// Mitsubishi GX Works2 project: Project - Done   PLC: FX3G

// global labels: Global1
VAR_GLOBAL
  startDay AT X007 : BOOL;
  startDayLamp AT Y007 : BOOL;
  amounts AT M0 : BOOL;
END_VAR
VAR_GLOBAL CONSTANT
  whippedCream : REAL := 300.0;
END_VAR
VAR_GLOBAL
  CreamTank AT D1105 : REAL;
END_VAR
VAR_GLOBAL CONSTANT
  Chocolate : REAL := 240;
  Chocolate_input : REAL := 240;
  whippedCream_input : REAL := 300;
END_VAR
VAR_GLOBAL
  ChocolateTank AT D1101 : REAL;
END_VAR
VAR_GLOBAL CONSTANT
  Biscuit_input : REAL := 6;
END_VAR
VAR_GLOBAL
  BiscuitTank AT D1103 : REAL;
  start_Proccessing AT X011 : BOOL;
END_VAR
VAR_GLOBAL CONSTANT
  Const_6 : REAL := 6;
END_VAR
VAR_GLOBAL
  binary_Less_than_6 AT M1 : BOOL;
END_VAR
VAR_GLOBAL CONSTANT
  Const_300 : REAL := 300;
END_VAR
VAR_GLOBAL
  binary_Less_than_300 AT M2 : BOOL;
END_VAR
VAR_GLOBAL CONSTANT
  Const_0 : REAL;
END_VAR
VAR_GLOBAL
  No_More_Raw AT M3 : BOOL;
  No_More_Raw_B AT M3 : BOOL;
  No_More_Raw_C AT M4 : BOOL;
  Proccess_B_Tank AT D1103 : REAL;
  Proccess_C_Tank AT D1104 : REAL;
  machine_A_On AT X010 : BOOL;
  machine_A_still_On AT M0 : BOOL;
  turn_machine_A_off AT X005 : BOOL;
  sen_Surface AT X001 : BOOL;
  sen_30 AT X002 : BOOL;
  sen_15 AT X003 : BOOL;
  currrently_sprinkling AT Y004 : BOOL;
  sen_camera AT X004 : BOOL;
END_VAR
VAR_GLOBAL CONSTANT
  TC0 : INT := 40;
  TC1 : INT := 40;
  constant_sec_4 : INT := 5;
END_VAR
VAR_GLOBAL
  time_total_4_sec_end_movement AT TC0 : BOOL;
  timer_ts0 AT TS0 : BOOL;
  lamp0 AT Y000 : BOOL;
  input_for_blinking AT M4 : BOOL;
  time_total_4_sec_end_movement2 AT TC1 : BOOL;
  timer_ts1 AT TS1 : BOOL;
  lamp1 AT Y001 : BOOL;
END_VAR
VAR_GLOBAL CONSTANT
  const_zero_val_word : INT;
END_VAR
VAR_GLOBAL
  analog_output AT D8282 : INT;
END_VAR
VAR_GLOBAL CONSTANT
  Const_240 : REAL := 240;
END_VAR
VAR_GLOBAL
  binary_Less_than_240 AT M3 : BOOL;
END_VAR
VAR_GLOBAL CONSTANT
  constant_4_sec : INT := 40;
END_VAR
VAR_GLOBAL
  time_total_4_sec_end_movement3 AT TC3 : BOOL;
END_VAR
VAR_GLOBAL CONSTANT
  constant_half_sec : INT := 5;
END_VAR
VAR_GLOBAL
  timer_ts3 AT TS3 : BOOL;
  start_Frosting AT X006 : BOOL;
  analog_Input_1 AT D8280 : INT;
  save_Analog_Value AT D1134 : INT;
  value_Sampled AT M10 : BOOL;
END_VAR
VAR_GLOBAL CONSTANT
  analog_upper_bound : INT := 3900;
  upper_bound_analog_value : INT := 3510;
  analog_lower_value : INT := 390;
END_VAR
VAR_GLOBAL
  input_is_invalid AT M11 : BOOL;
  currently_frosting AT Y003 : BOOL;
END_VAR
VAR_GLOBAL CONSTANT
  single_frosting_check : INT := 1950;
END_VAR
VAR_GLOBAL
  single_frosting AT M12 : BOOL;
  double_frosting AT M13 : BOOL;
END_VAR
VAR_GLOBAL CONSTANT
  chocalate_single_amount : INT := 120;
END_VAR
VAR_GLOBAL
  dipping_tank AT D1107 : REAL;
END_VAR
VAR_GLOBAL CONSTANT
  chocalate_double_amount : INT := 240;
END_VAR
VAR_GLOBAL
  frostimg_time AT TC5 : BOOL;
END_VAR
VAR_GLOBAL CONSTANT
  const_5_sec : INT := 50;
END_VAR
VAR_GLOBAL
  frosting_time_over AT TS5 : BOOL;
END_VAR
VAR_GLOBAL CONSTANT
  const_chocalate_single_amount : REAL := 120;
  const_chocalate_double_amount : REAL := 240;
END_VAR
VAR_GLOBAL
  analog_Input_2 AT D8281 : INT;
  start_Packing AT X011 : BOOL;
END_VAR
VAR_GLOBAL CONSTANT
  const_count_5 : INT := 5;
END_VAR
VAR_GLOBAL
  start_packing_counter AT CC1 : BOOL;
  finish_packing_5_counter AT CS1 : BOOL;
  packing_5_lamp AT Y002 : BOOL;
  end_of_movment AT M20 : BOOL;
  pack_one_krembo AT X000 : BOOL;
  finish_packing_counter AT CC2 : BOOL;
END_VAR
VAR_GLOBAL CONSTANT
  const_count_1 : INT := 1;
END_VAR
VAR_GLOBAL
  finish_packing_6_counter AT CS3 : BOOL;
  finish_packing_1_counter AT CS2 : BOOL;
  finish_total_packing_counter AT CC3 : BOOL;
END_VAR
VAR_GLOBAL CONSTANT
  const_count_6 : INT := 6;
END_VAR
VAR_GLOBAL
  finish_packing_all_counter AT CS3 : BOOL;
  Proccess_Cream_Tank AT D1109 : REAL;
  Proccess_chocolate_tank AT D1107 : REAL;
  end_of_packing AT M22 : BOOL;
END_VAR
VAR_GLOBAL CONSTANT
  Const_6_krembos : REAL := 240;
END_VAR
VAR_GLOBAL
  krembo_total_count AT D10 : REAL;
  word_krembo_total AT D1150 : INT;
END_VAR
VAR_GLOBAL CONSTANT
  Const_6_x : REAL := 2340;
END_VAR
VAR_GLOBAL
  double_frosting_lamp AT M100 : BOOL;
  stsrt_frosting_lamp AT M21 : BOOL;
  start_frosting_lamp AT M21 : BOOL;
  frosting AT M34 : BOOL;
  krembo_added AT M40 : BOOL;
  less_Than_6 AT M41 : BOOL;
  cream_less_than_300 AT M42 : BOOL;
  chocolate_less_than_240 AT M43 : BOOL;
  biscuit_less_Than_6 AT M41 : BOOL;
END_VAR
VAR_GLOBAL CONSTANT
  double_frosting_check : INT := 2340;
END_VAR
VAR_GLOBAL
  converted AT M45 : BOOL;
  time_total_3_sec_end_day : BOOL;
  time_total_3_sec_end_day2 : BOOL;
  timer_ts100 : BOOL;
  timer_ts101 : BOOL;
  const_3_sec_timer AT TC6 : BOOL;
END_VAR
VAR_GLOBAL CONSTANT
  const_3_sec : INT := 30;
END_VAR
VAR_GLOBAL
  time_3_sec AT TC6 : BOOL;
  timer_ts_6 AT TS6 : BOOL;
  time_3_sec_end_day AT TC7 : BOOL;
  day_over_lamp AT M46 : BOOL;
  day_over AT M46 : BOOL;
  timer_ts_7 AT TS7 : BOOL;
  time_3_sec_end_day2 AT TC8 : BOOL;
  end_Day_Blink AT M50 : BOOL;
  timer_ts_8 AT TS8 : BOOL;
  fake_light AT M51 : BOOL;
  input_for_end_day_blink AT M60 : BOOL;
  flick_time_still AT M70 : BOOL;
  flicker_end_day AT M71 : BOOL;
  blink_1 AT M72 : BOOL;
  tc_blink1 AT TC9 : BOOL;
END_VAR
VAR_GLOBAL CONSTANT
  const_quick_3 : INT := 5;
END_VAR
VAR_GLOBAL
  ts_blink1 AT TS9 : BOOL;
  za_blink1 AT M73 : BOOL;
  tc_blink2 AT TC10 : BOOL;
  ts_blink10 AT TS10 : BOOL;
  za_blink2 AT M74 : BOOL;
  ts_blink2 AT TS10 : BOOL;
END_VAR

// task Task_01 (event TRUE, interval 0, priority 31): POU_01

PROGRAM POU_01
VAR
  timer_ts6 : BOOL;
END_VAR
(* structured ladder/FBD written out as ST: instructions are called as NAME(EN, inputs, outputs); _pN, _eN, _tN stand for wires *)
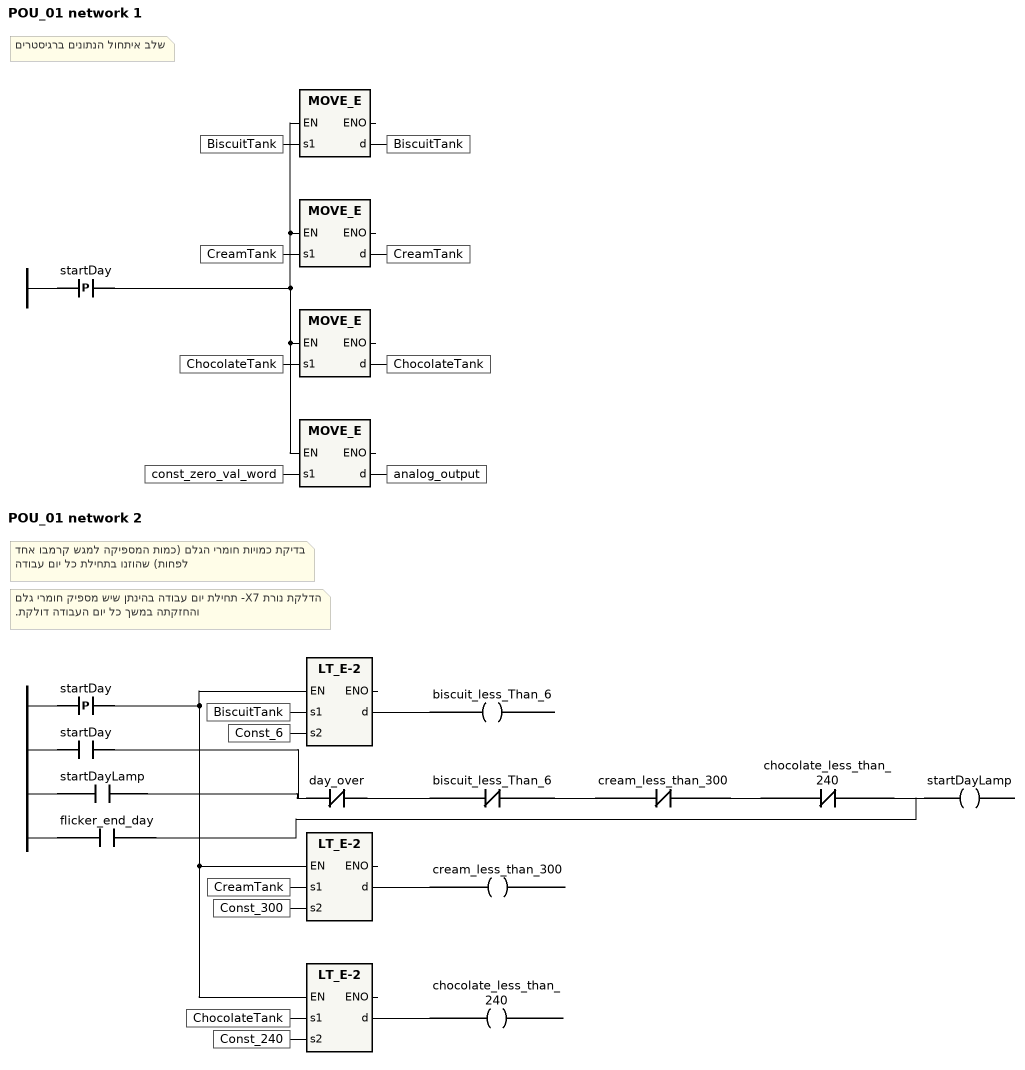
(* network 1 User input *)
(* שלב איתחול הנתונים ברגיסטרים *)
_p1 := LDP(TRUE, startDay);
MOVE_E(_p1, BiscuitTank, BiscuitTank);
MOVE_E(_p1, CreamTank, CreamTank);
MOVE_E(_p1, ChocolateTank, ChocolateTank);
MOVE_E(_p1, const_zero_val_word, analog_output);
(* network 2 Day initialize *)
(* בדיקת כמויות חומרי הגלם (כמות המספיקה למגש קרמבו אחד לפחות) שהוזנו בתחילת כל יום עבודה *)
(* הדלקת נורת X7- תחילת יום עבודה בהינתן שיש מספיק חומרי גלם והחזקתה במשך כל יום העבודה דולקת. *)
_p1 := LDP(TRUE, startDay);
LT_E(_p1, BiscuitTank, Const_6, _t2);
biscuit_less_Than_6 := _t2;
LT_E(_p1, CreamTank, Const_300, _t3);
cream_less_than_300 := _t3;
LT_E(_p1, ChocolateTank, Const_240, _t4);
chocolate_less_than_240 := _t4;
startDayLamp := (((((startDay OR startDayLamp) AND NOT day_over) AND NOT biscuit_less_Than_6) AND NOT cream_less_than_300) AND NOT chocolate_less_than_240) OR flicker_end_day;
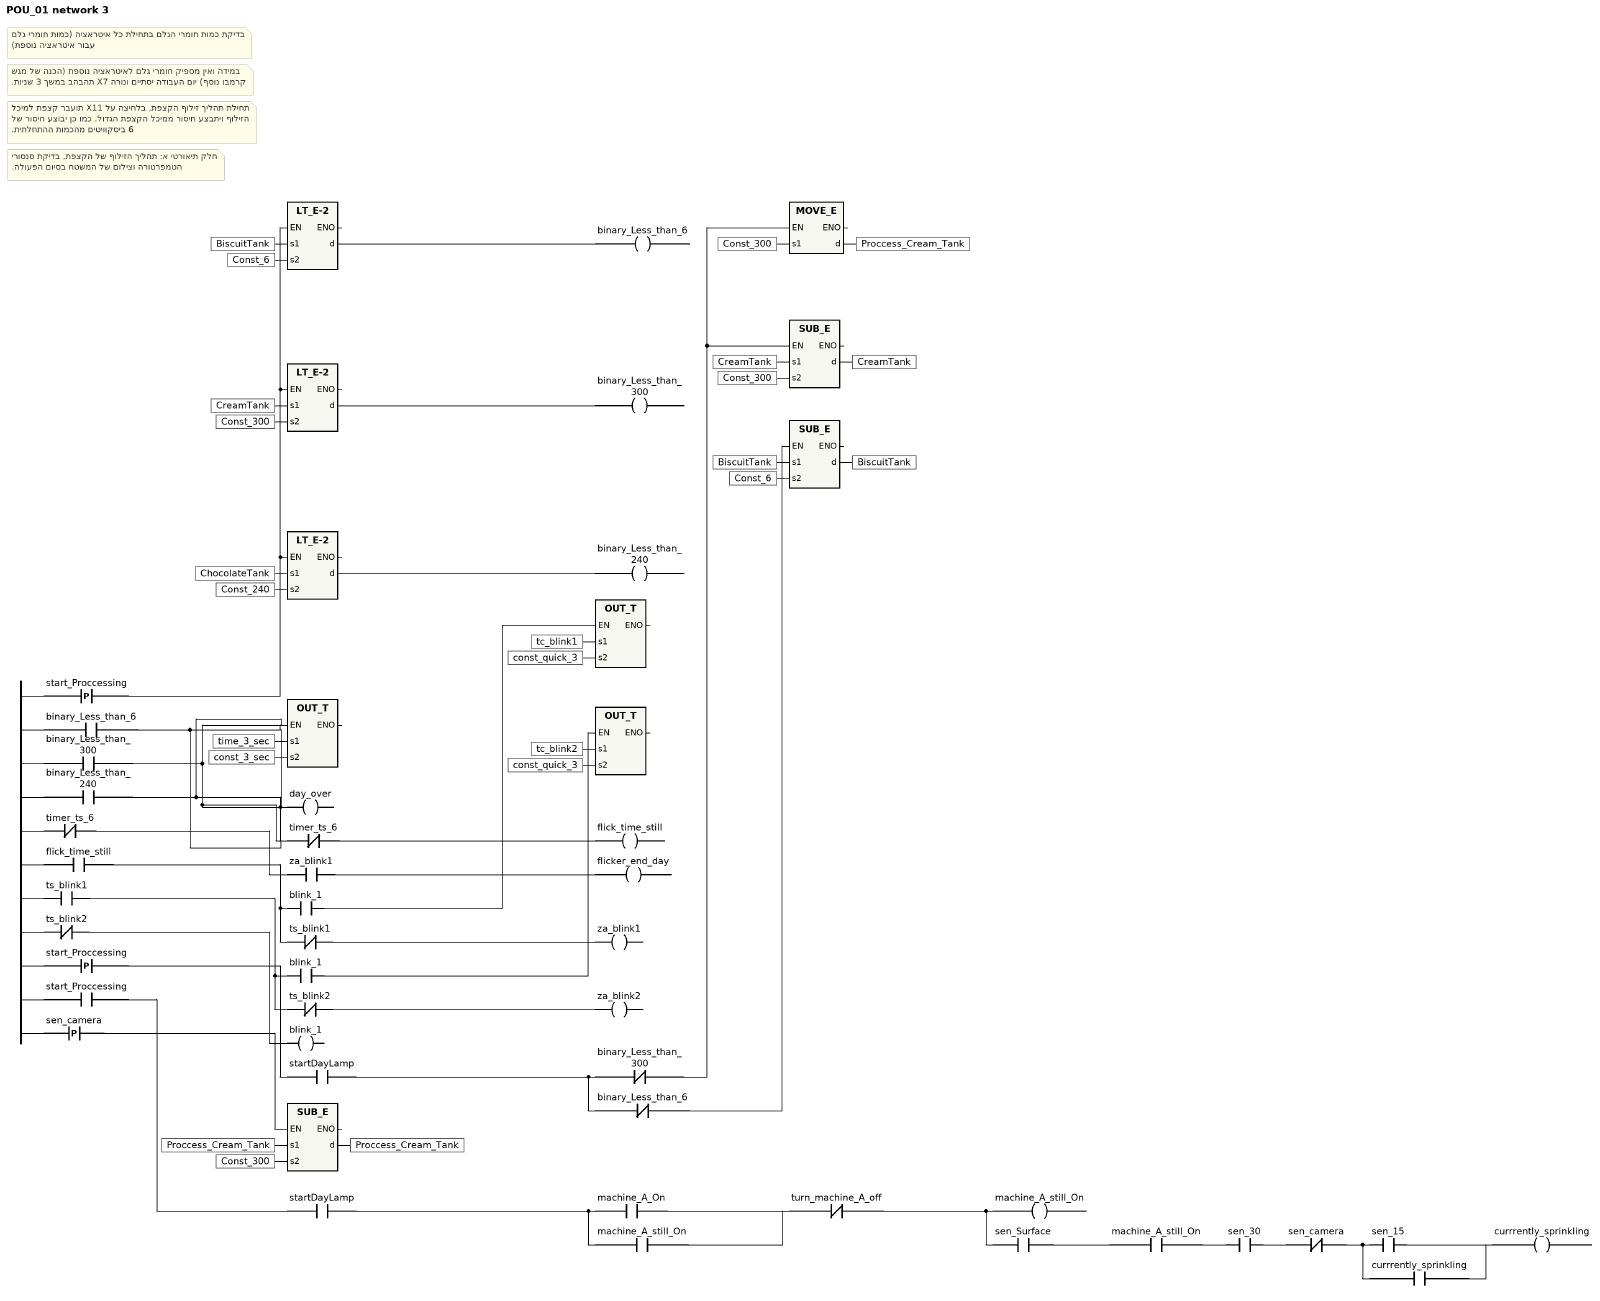
(* network 3 Whipping Cream Proc *)
(* בדיקת כמות חומרי הגלם בתחילת כל איטראציה (כמות חומרי גלם עבור איטראציה נוספת) *)
(* במידה ואין מספיק חומרי גלם לאיטראציה נוספת (הכנה של מגש קרמבו נוסף) יום העבודה יסתיים ונורה X7 תהבהב במשך 3 שניות. *)
(* תחילת תהליך זילוף הקצפת, בלחיצה על X11 תועבר קצפת למיכל הזילוף ויתבצע חיסור ממיכל הקצפת הגדול. כמו כן יבוצע חיסור של 6 ביסקוויטים מהכמות ההתחלתית. *)
(* חלק תיאורטי א: תהליך הזילוף של הקצפת, בדיקת סנסורי הטמפרטורה וצילום של המשטח בסיום הפעולה. *)
_p1 := LDP(TRUE, start_Proccessing);
LT_E(_p1, BiscuitTank, Const_6, _t2);
binary_Less_than_6 := _t2;
LT_E(_p1, CreamTank, Const_300, _t3);
binary_Less_than_300 := _t3;
LT_E(_p1, ChocolateTank, Const_240, _t4);
binary_Less_than_240 := _t4;
_p5 := binary_Less_than_6 OR binary_Less_than_300 OR binary_Less_than_240;
OUT_T(_p5, time_3_sec, const_3_sec);
day_over := _p5;
flick_time_still := _p5 AND NOT timer_ts_6;
flicker_end_day := NOT timer_ts_6 AND za_blink1;
OUT_T(flick_time_still AND blink_1, tc_blink1, const_quick_3);
za_blink1 := flick_time_still AND NOT ts_blink1;
OUT_T(ts_blink1 AND blink_1, tc_blink2, const_quick_3);
za_blink2 := ts_blink1 AND NOT ts_blink2;
blink_1 := NOT ts_blink2;
_p6 := LDP(TRUE, start_Proccessing) AND startDayLamp;
_p7 := _p6 AND NOT binary_Less_than_300;
MOVE_E(_p7, Const_300, Proccess_Cream_Tank);
SUB_E(_p7, CreamTank, Const_300, CreamTank);
SUB_E(_p6 AND NOT binary_Less_than_6, BiscuitTank, Const_6, BiscuitTank);
_p8 := start_Proccessing AND startDayLamp;
_p9 := ((_p8 AND machine_A_On) OR (_p8 AND machine_A_still_On)) AND NOT turn_machine_A_off;
machine_A_still_On := _p9;
_p10 := _p9 AND sen_Surface AND machine_A_still_On AND sen_30 AND NOT sen_camera;
currrently_sprinkling := (_p10 AND sen_15) OR (_p10 AND currrently_sprinkling);
SUB_E(LDP(TRUE, sen_camera), Proccess_Cream_Tank, Const_300, Proccess_Cream_Tank);
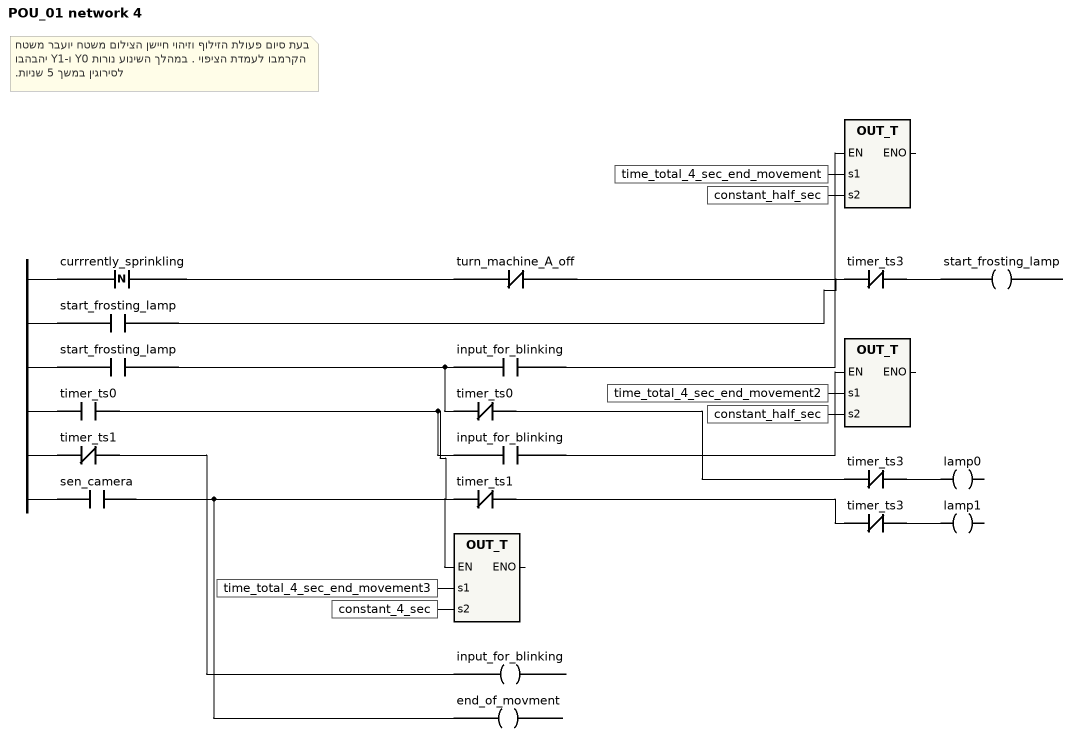
(* network 4 Move the krembo to B *)
(* בעת סיום פעולת הזילוף וזיהוי חיישן הצילום משטח יועבר משטח הקרמבו לעמדת הציפוי . במהלך השינוע נורות Y0 ו-Y1 יהבהבו לסירוגין במשך 5 שניות. *)
start_frosting_lamp := ((LDF(TRUE, currrently_sprinkling) AND NOT turn_machine_A_off) OR start_frosting_lamp) AND NOT timer_ts3;
OUT_T(start_frosting_lamp AND input_for_blinking, time_total_4_sec_end_movement, constant_half_sec);
lamp0 := start_frosting_lamp AND NOT timer_ts0 AND NOT timer_ts3;
OUT_T(timer_ts0 AND input_for_blinking, time_total_4_sec_end_movement2, constant_half_sec);
lamp1 := timer_ts0 AND NOT timer_ts1 AND NOT timer_ts3;
input_for_blinking := NOT timer_ts1;
OUT_T(sen_camera, time_total_4_sec_end_movement3, constant_4_sec);
end_of_movment := sen_camera;
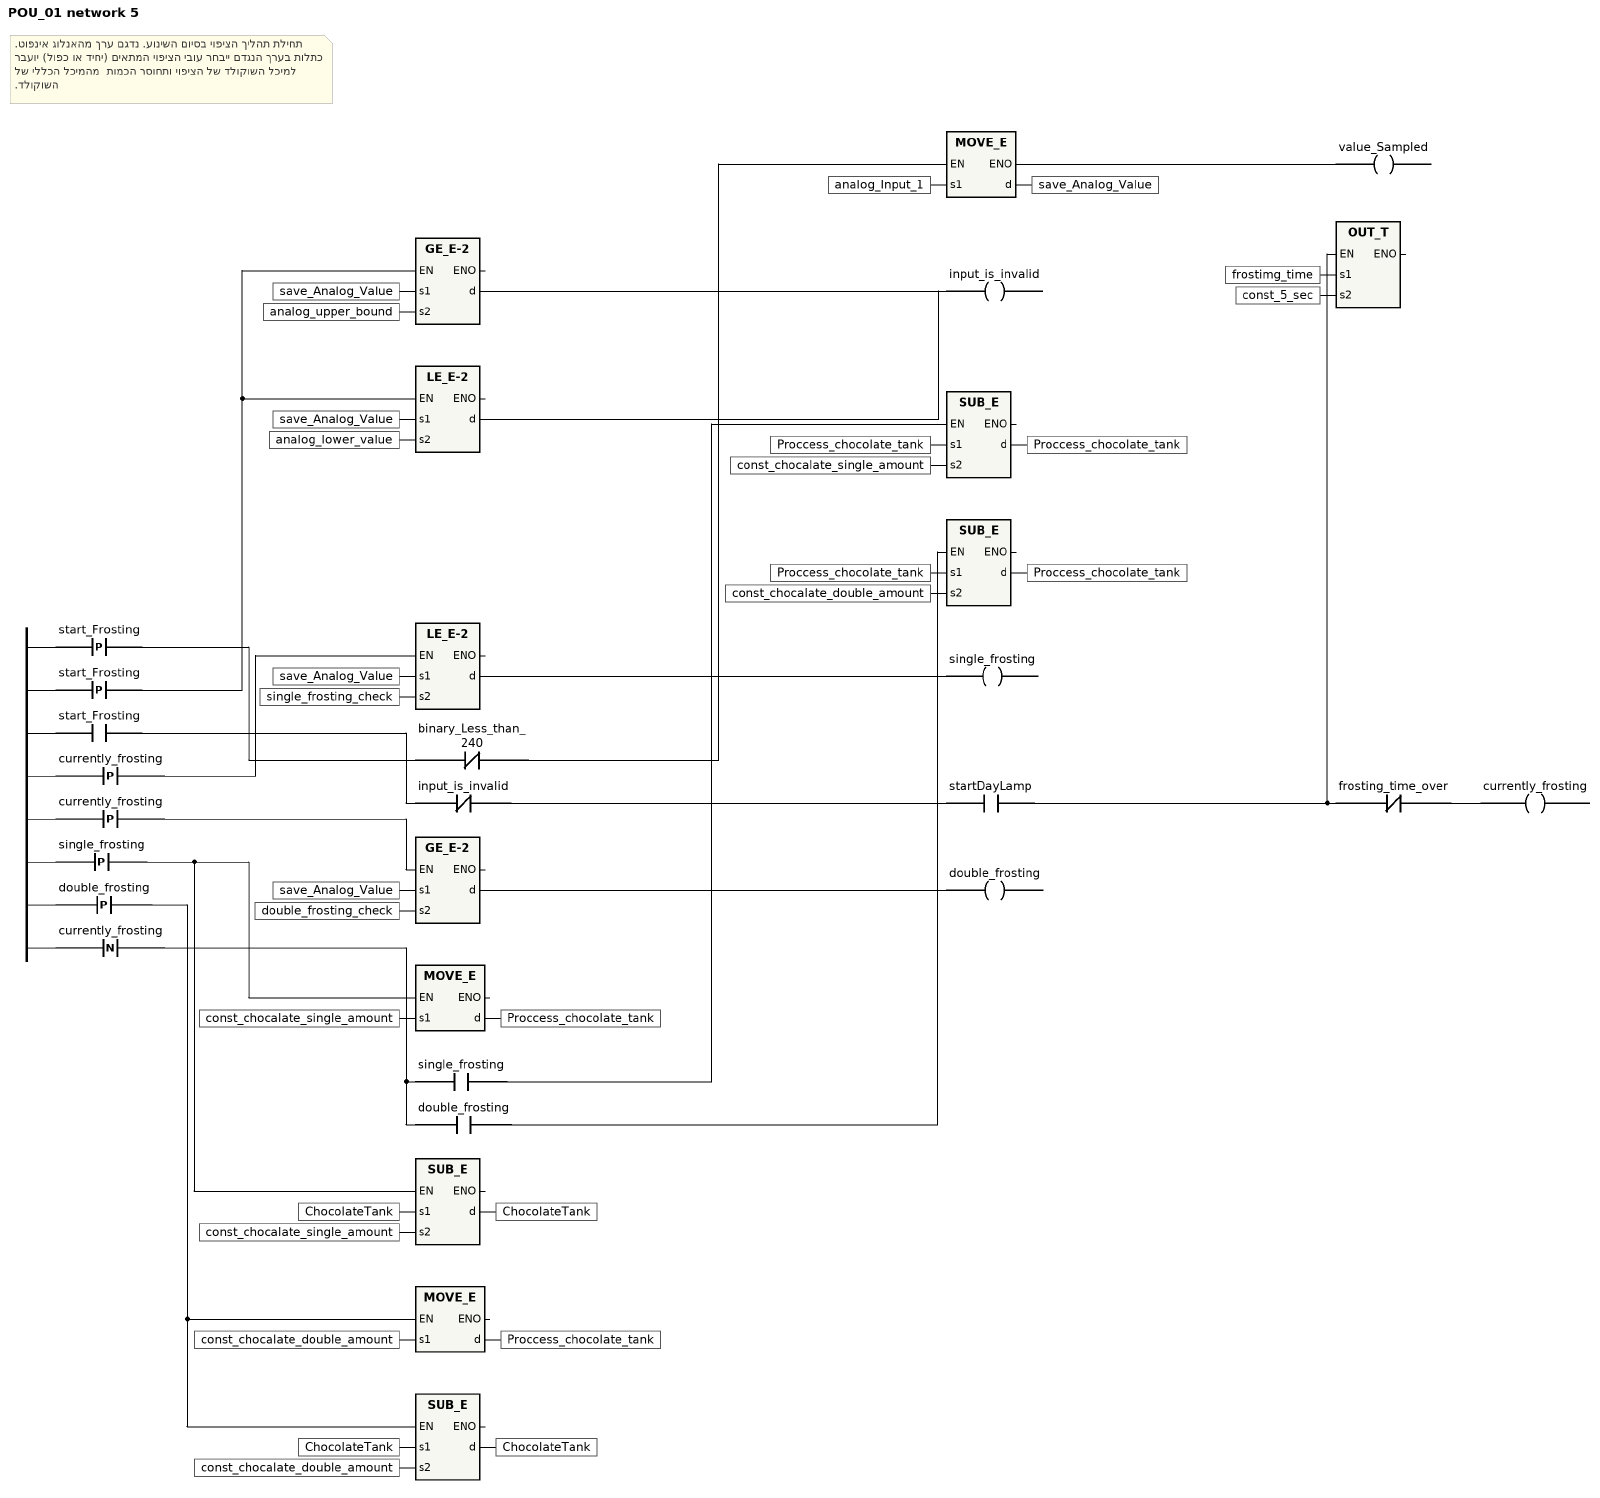
(* network 5 Frosting *)
(* תחילת תהליך הציפוי בסיום השינוע. נדגם ערך מהאנלוג אינפוט. כתלות בערך הנגדם ייבחר עובי הציפוי המתאים (יחיד או כפול) יועבר למיכל השוקולד של הציפוי ותחוסר הכמות  מהמיכל הכללי של השוקולד. *)
_e1 := MOVE_E(LDP(TRUE, start_Frosting) AND NOT binary_Less_than_240, analog_Input_1, save_Analog_Value);
value_Sampled := _e1;
_p2 := LDP(TRUE, start_Frosting);
GE_E(_p2, save_Analog_Value, analog_upper_bound, _t3);
LE_E(_p2, save_Analog_Value, analog_lower_value, _t4);
input_is_invalid := _t3 OR _t4;
_p5 := start_Frosting AND NOT input_is_invalid AND startDayLamp;
OUT_T(_p5, frostimg_time, const_5_sec);
currently_frosting := _p5 AND NOT frosting_time_over;
LE_E(LDP(TRUE, currently_frosting), save_Analog_Value, single_frosting_check, _t6);
single_frosting := _t6;
GE_E(LDP(TRUE, currently_frosting), save_Analog_Value, double_frosting_check, _t7);
double_frosting := _t7;
_p8 := LDP(TRUE, single_frosting);
MOVE_E(_p8, const_chocalate_single_amount, Proccess_chocolate_tank);
SUB_E(_p8, ChocolateTank, const_chocalate_single_amount, ChocolateTank);
_p9 := LDP(TRUE, double_frosting);
MOVE_E(_p9, const_chocalate_double_amount, Proccess_chocolate_tank);
SUB_E(_p9, ChocolateTank, const_chocalate_double_amount, ChocolateTank);
_p10 := LDF(TRUE, currently_frosting);
SUB_E(_p10 AND single_frosting, Proccess_chocolate_tank, const_chocalate_single_amount, Proccess_chocolate_tank);
SUB_E(_p10 AND double_frosting, Proccess_chocolate_tank, const_chocalate_double_amount, Proccess_chocolate_tank);
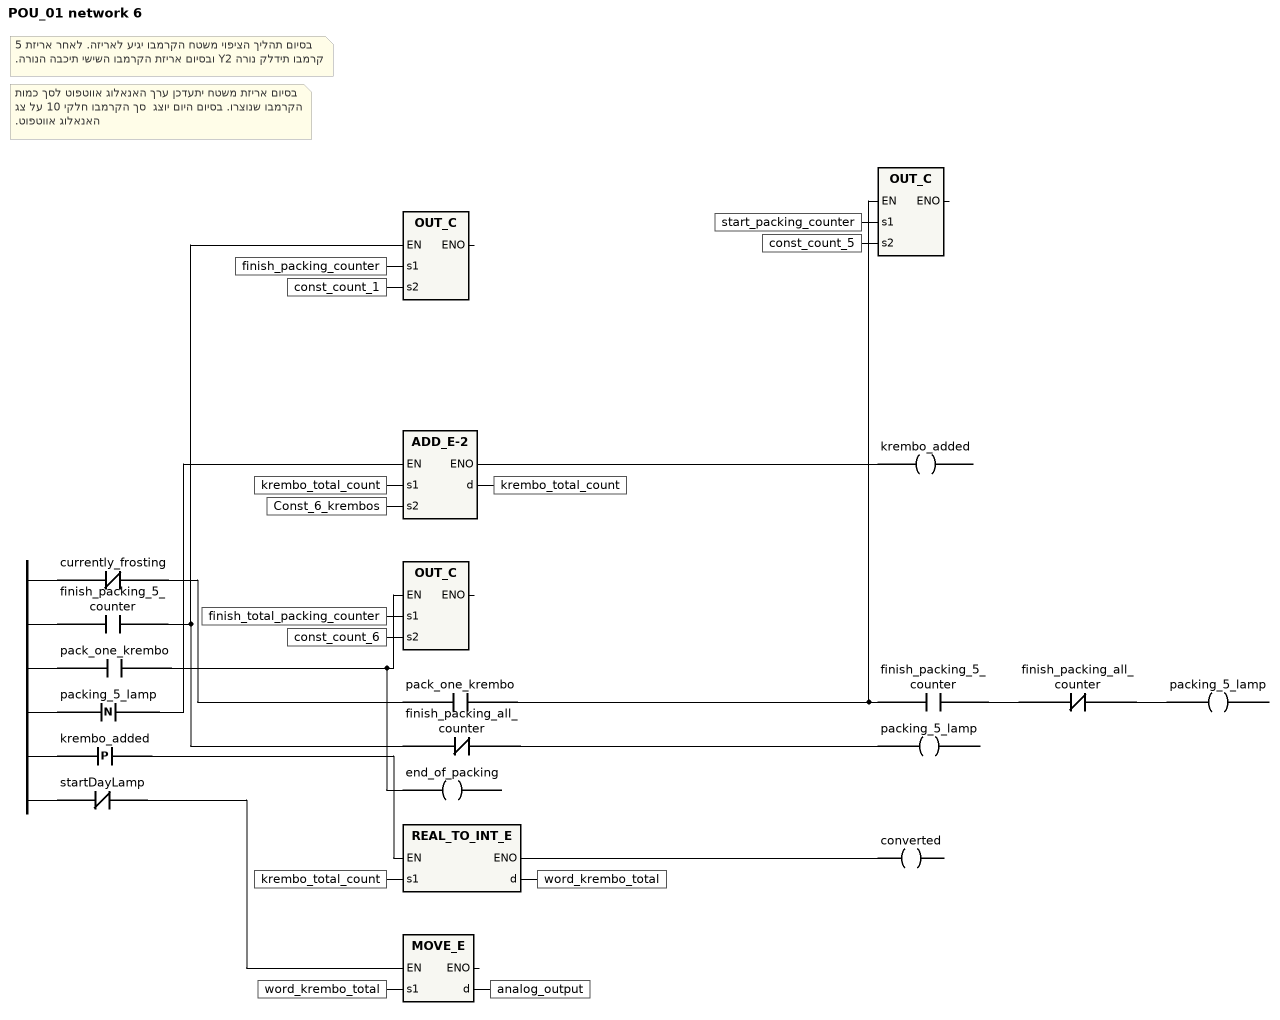
(* network 6 packing krembo *)
(* בסיום תהליך הציפוי משטח הקרמבו יגיע לאריזה. לאחר אריזת 5 קרמבו תידלק נורה Y2 ובסיום אריזת הקרמבו השישי תיכבה הנורה. *)
(* בסיום אריזת משטח יתעדכן ערך האנאלוג אווטפוט לסך כמות הקרמבו שנוצרו. בסיום היום יוצג  סך הקרמבו חלקי 10 על צג האנאלוג אווטפוט. *)
_p1 := NOT currently_frosting AND pack_one_krembo;
OUT_C(_p1, start_packing_counter, const_count_5);
packing_5_lamp := _p1 AND finish_packing_5_counter AND NOT finish_packing_all_counter;
OUT_C(finish_packing_5_counter, finish_packing_counter, const_count_1);
packing_5_lamp := finish_packing_5_counter AND NOT finish_packing_all_counter;
OUT_C(pack_one_krembo, finish_total_packing_counter, const_count_6);
end_of_packing := pack_one_krembo;
_e2 := ADD_E(LDF(TRUE, packing_5_lamp), krembo_total_count, Const_6_krembos, krembo_total_count);
krembo_added := _e2;
_e3 := REAL_TO_INT_E(LDP(TRUE, krembo_added), krembo_total_count, word_krembo_total);
converted := _e3;
MOVE_E(NOT startDayLamp, word_krembo_total, analog_output);
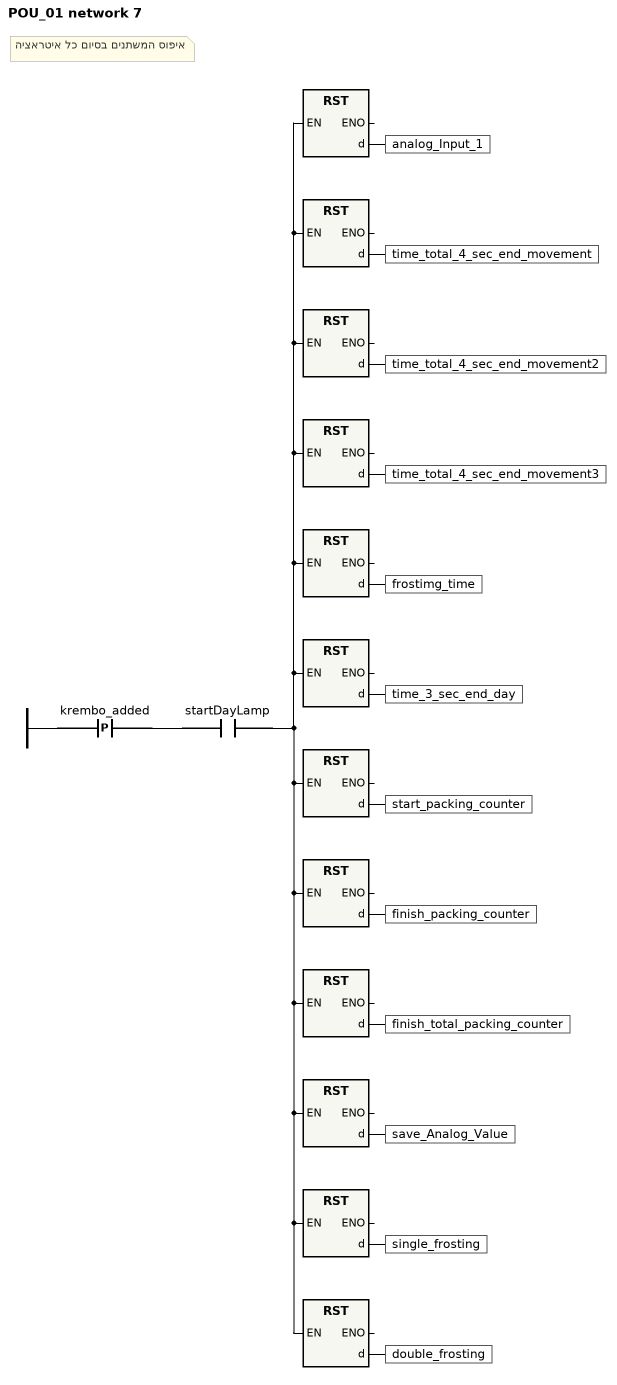
(* network 7 reset *)
(* איפוס המשתנים בסיום כל איטראציה *)
_p1 := LDP(TRUE, krembo_added) AND startDayLamp;
RST(_p1, analog_Input_1);
RST(_p1, time_total_4_sec_end_movement);
RST(_p1, time_total_4_sec_end_movement2);
RST(_p1, time_total_4_sec_end_movement3);
RST(_p1, frostimg_time);
RST(_p1, time_3_sec_end_day);
RST(_p1, start_packing_counter);
RST(_p1, finish_packing_counter);
RST(_p1, finish_total_packing_counter);
RST(_p1, save_Analog_Value);
RST(_p1, single_frosting);
RST(_p1, double_frosting);
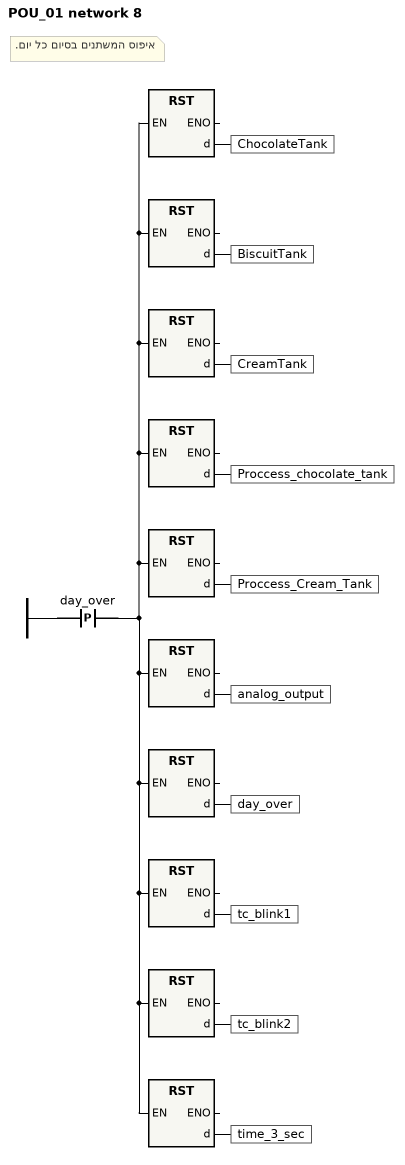
(* network 8 *)
(* איפוס המשתנים בסיום כל יום. *)
_p1 := LDP(TRUE, day_over);
RST(_p1, ChocolateTank);
RST(_p1, BiscuitTank);
RST(_p1, CreamTank);
RST(_p1, Proccess_chocolate_tank);
RST(_p1, Proccess_Cream_Tank);
RST(_p1, analog_output);
RST(_p1, day_over);
RST(_p1, tc_blink1);
RST(_p1, tc_blink2);
RST(_p1, time_3_sec);
END_PROGRAM
